// TIA Portal V20 export
DATA_BLOCK "LPFE_MonitorData"   // DB245
{ DB_Accessible_From_OPC_UA := 'FALSE' }
// stored: Access Published, DBAccessibleFromOPCUA false, DBAccessibleFromWebserver false, MemoryReserve 100, Namespace PFE
   VAR
      Channels : Array[0.._.LE_NUMBER_OF_INTERFACE_BUFFERS] of "LPFE_typeDiagnosticMonitorChannel";
      Transactions : Array[0.._.SIZE_TRANSACTIONS_ARRAY] of "LPFE_typePFEData";
      healthData : "LPFE_typeMonitorData";
      shiftElapsedTime { S7_SetPoint := 'True'} : Time;   // Shift's elapsed time after reinitialization
      newTransactions { S7_SetPoint := 'True'} : Int;   // New processed Transactions
   END_VAR
BEGIN
END_DATA_BLOCK
